// TIA Portal V17 export
// export: Created 2024-09-02T12:50:29.0385036Z, ExportSetting WithDefaults, DisplayName Totally Integrated Automation Portal, DisplayVersion V17, DisplayName TIA Portal Openness, DisplayVersion V17, DisplayName TIA Portal Version Control Interface, DisplayVersion V17, DisplayName STEP 7 Professional, DisplayVersion V17, DisplayName STEP 7 Safety, DisplayVersion V17, DisplayName WinCC Professional, DisplayVersion V17
TYPE "TypeProcessScreen"
// stored: IsFailsafeCompliant false
   STRUCT
      STAT : Struct
         TOTAL_OK : Bool;
         TOTAL_NOK : Bool;
         CHOICE_AVAILABLE : Bool;
         HAND_OK_AVAILABLE : Bool;
         REWORK_AVAILABLE : Bool;
         NOK_REJECT : Bool;
         REPEAT_AFTER_NOK : Bool;
         NOK_AVAILABLE : Bool;
      END_STRUCT;
      Process : Struct
         PROC_NR : Int;   // TAF NR / TAF NR
         Status : Int;   // 1=IO; 2=NIO / 1 = OK, 2 = NOK
         DES : Array[1..22] of Char;   // Bezeichnung / Description
      END_STRUCT;
      BUTTON_REPEAT_NOK : Struct   // Taste Wiederholen nach NIO / Repeat button to NOK
         fade_in : Bool;   // Taste einblenden / Show button
         operated : Bool;   // Taste wurde betaetigt / Button was pressed
         executable : Bool;   // Taste ist Ausführbar Schrift sw / Button is executable Font sw
         function_active : Bool;   // Funktion ist aktiv / Function is active
         Formation : Int;   // Gestaltung Taste / Design button
      END_STRUCT;
      BUTTON_NOK_RELEASE : Struct   // Taste NIO Entlassen / Approve NOK Button
         fade_in : Bool;   // Taste einblenden / Show button
         operated : Bool;   // Taste wurde betaetigt / Button was pressed
         executable : Bool;   // Taste ist Ausführbar Schrift sw / Button is executable Font sw
         function_active : Bool;   // Funktion ist aktiv / Function is active
         Formation : Int;   // Gestaltung Taste / Design button
      END_STRUCT;
      BUTTON_SD_OPEN : Struct   // Taste Schutztür entriegeln / Unlock safety door button
         fade_in : Bool;   // Taste einblenden / Show button
         operated : Bool;   // Taste wurde betaetigt / Button was pressed
         executable : Bool;   // Taste ist Ausführbar Schrift sw / Button is executable Font sw
         function_active : Bool;   // Funktion ist aktiv / Function is active
         Formation : Int;   // Gestaltung Taste / Design button
      END_STRUCT;
      BUTTON_SD_CLOSE : Struct   // Taste Schutztür verriegeln / Lock safety door button
         fade_in : Bool;   // Taste einblenden / Show button
         operated : Bool;   // Taste wurde betaetigt / Button was pressed
         executable : Bool;   // Taste ist Ausführbar Schrift sw / Button is executable Font sw
         function_active : Bool;   // Funktion ist aktiv / Function is active
         Formation : Int;   // Gestaltung Taste / Design button
      END_STRUCT;
      GENERAL : Struct
         Lamp_Nr : Int;   // Ampelnummer / Lamp number
      END_STRUCT;
      EDIT : Struct
         Lamp_Nr : Int;   // Ampelnummer / Lamp number
         active : Bool;   // Editierdialog aktiv / Editing dialog active
         BUTTON_DESELECTION : Struct   // Taste Abwahl / Deselect button
            fade_in : Bool;   // Taste einblenden / Show button
            operated : Bool;   // Taste wurde betaetigt / Button was pressed
            executable : Bool;   // Taste ist Ausführbar Schrift sw / Button is executable Font sw
            function_active : Bool;   // Funktion ist aktiv / Function is active
            Formation : Int;   // Gestaltung Taste / Design button
         END_STRUCT;
         BUTTON_HAND_OK : Struct   // Taste Hand IO / Manual button OK
            fade_in : Bool;   // Taste einblenden / Show button
            operated : Bool;   // Taste wurde betaetigt / Button was pressed
            executable : Bool;   // Taste ist Ausführbar Schrift sw / Button is executable Font sw
            function_active : Bool;   // Funktion ist aktiv / Function is active
            Formation : Int;   // Gestaltung Taste / Design button
         END_STRUCT;
         BUTTON_ACCEPT : Struct   // Taste Übernehmen / Apply button
            fade_in : Bool;   // Taste einblenden / Show button
            operated : Bool;   // Taste wurde betaetigt / Button was pressed
            executable : Bool;   // Taste ist Ausführbar Schrift sw / Button is executable Font sw
            function_active : Bool;   // Funktion ist aktiv / Function is active
            Formation : Int;   // Gestaltung Taste / Design button
         END_STRUCT;
         BUTTON_CANCEL : Struct   // Taste Abbrechen / Cancel button
            fade_in : Bool;   // Taste einblenden / Show button
            operated : Bool;   // Taste wurde betaetigt / Button was pressed
            executable : Bool;   // Taste ist Ausführbar Schrift sw / Button is executable Font sw
            function_active : Bool;   // Funktion ist aktiv / Function is active
            Formation : Int;   // Gestaltung Taste / Design button
         END_STRUCT;
      END_STRUCT;
      LAMP : Array[1..64] of Struct
         fade_in : Bool;   // Symbol einblenden / Show symbol
         colour : Int;   // Farbe für HMI 1=Gelb/blink; 2=Gelb;3=Grün;4=Blau;5=Rot;6=Hellgrün / Color for HMI 1=Yellow/blink; 2=Yellow;3=Green;4=Blue;5=Red;6=Light green
      END_STRUCT;
      D : Struct
         STATUS : Struct
            LP_HAS_WORKED : Bool;   // Status der letzten Bearbeitung: Station hat gearbeitet / Status of last processing: Station has worked
            LP_HAS_OK_WORKED : Bool;   // Status der letzten Bearbeitung: Station hat Io. gearbeitet / Status of last processing: Station has worked OK
            LP_HAS_NOK_WORKED : Bool;   // Status der letzten Bearbeitung: Station hat Nio. gearbeitet / Status of last processing: Station has worked NOK
            LP_HAS_WORKED_WITH_DESEL : Bool;   // Status der letzten Bearbeitung: Station hat gearbeitet mit abgewählt / Status of last processing: Station has worked with deselected
            LP_HAS_WORKED_WITH_HAND_OK : Bool;   // Status der letzten Bearbeitung: Station hat gearbeitet mit Hand Io. / Status of last machining: Station has worked with manual OK
            LP_BIT_0_5 : Bool;   // Status der letzten Bearbeitung: / Status of the last processing:
            LP_BIT_0_6 : Bool;   // Status der letzten Bearbeitung: / Status of the last processing:
            LP_BIT_0_7 : Bool;   // Status der letzten Bearbeitung: / Status of the last processing:
            FP_HAS_WORKED : Bool;   // Status der ersten Bearbeitung: Station hat gearbeitet / Status of first processing: Station has worked
            FP_HAS_OK_WORKED : Bool;   // Status der ersten Bearbeitung: Station hat Io. gearbeitet / Status of first processing: Station has worked OK
            FP_HAS_NOK_WORKED : Bool;   // Status der ersten Bearbeitung: Station hat Nio. gearbeitet / Status of first processing: Station has worked NOK
            FP_HAS_WORKED_WITH_DESEL : Bool;   // Status der ersten Bearbeitung: Station hat gearbeitet mit abgewählt / Status of first processing: Station has worked with deselected
            FP_HAS_WORKED_WITH_HAND_OK : Bool;   // Status der ersten Bearbeitung: Station hat gearbeitet mit Hand Io. / Status of first machining: Station has worked with hand OK
            FP_BIT_0_5 : Bool;   // Status der ersten Bearbeitung: / Status of the first processing:
            FP_BIT_0_6 : Bool;   // Status der ersten Bearbeitung: / Status of the first processing:
            FP_BIT_0_7 : Bool;   // Status der ersten Bearbeitung: / Status of the first processing:
            PASS_COUNTER : Byte;
            BLOCKCHECK : Byte;
         END_STRUCT;
         GRP_BUSY : Array[0..7] of Bool;   // Gruppe belegt / Group occupied
         GRP_OK : Array[0..7] of Bool;   // Gruppe i.O. / Group OK
         GRP_NOK : Array[0..7] of Bool;   // Gruppe n.i.O. / Group NOK
         GRP_DESELECTED : Array[0..7] of Bool;   // Gruppe abgewählt / Group deselected
         GRP_HAND_OK : Array[0..7] of Bool;   // Gruppe Hand i.O. / Group Hand OK
         GRP : Array[0..7] of Struct
            EZB_Loaded : Array[0..7] of Bool;   // Einzelbearbeitung belegt / Individual processing occupied
            EZB_OK : Array[0..7] of Bool;   // Einzelbearbeitung i.O. / Individual processing OK
            EZB_NOK : Array[0..7] of Bool;   // Einzelbearbeitung n.i.O. / Individual processing NOK
            EZB_Deselected : Array[0..7] of Bool;   // Einzelbearbeitung abgewählt / Individual processing deselected
            EZB_HAND_OK : Array[0..7] of Bool;   // Einzelbearbeitung Hand i.O. / Individual machining hand OK
            Continuous_Counter : Byte;
         END_STRUCT;
         STATION_WORK_YEAR : Byte;
         STATION_WORK_MONTH : Byte;
         STATION_WORK_DAY : Byte;
         STATION_WORK_HOUR : Byte;
         STATION_WORK_MINUTE : Byte;
         STATION_WORK_SECOND : Byte;
         WORKER_ID : DWord;
      END_STRUCT;
      WorkInstr : Struct   // Arbeitsanweisung / Working instruction
         MP_Nr : Array[1..16] of Int;   // Anzeige MP / Display MP
         Intern : Struct
            Pointer : Int := 1;
            Index : Array[1..16] of Int;   // Index
         END_STRUCT;
      END_STRUCT;
      ABWAHL_EXT { ExternalWritable := 'False'} : Array[1..64] of Bool;
   END_STRUCT;
END_TYPE
